(* IEC 61131-3 sources: stverif/testfiles, 5 files *)

(* ---- test.typ ---- *)
TYPE
	My_Struct : STRUCT
		out : INT;
	END_STRUCT;
    Valve : STRUCT
        Value : REAL;
    END_STRUCT;
END_TYPE

(* ---- test.fun ---- *)
FUNCTION I_TO_R : REAL
    VAR_INPUT
        IN : INT;
    END_VAR
END_FUNCTION

(* ---- test.st ---- *)
PROGRAM name_this_program_pls

	// Initialize ControlValues

	FOR n := 1 TO 16 DO
	    k := (45.0 * (k + I_TO_R(n))) / 1000.0;
	END_FOR

	CtrlLEFT  := k;
	CtrlRIGHT := k;

	// Case from the ControlValue with Controller logic action call
  CASE k OF
      1,3,7   :   CtrlLEFT  := a;
      4,6     :   CtrlRIGHT := b;
      ELSE        PosForceCtrl;
  END_CASE

	// Map controller output to hardware
	IF enableCtrlValves.out THEN
	    RightValve.Value    := CtrlLEFT;
	    LeftValve.Value        := CtrlRIGHT;
	ELSE
      ValveCtrl := 0;
  END_IF
END_PROGRAM

(* ---- test.var ---- *)
VAR
    n : INT;
    k : REAL;
    a : REAL;
    b : REAL;
    CtrlLEFT : REAL;
    CtrlRIGHT : REAL;
    enableCtrlValves : My_Struct;
    RightValve : Valve;
    LeftValve : Valve;
    ValveCtrl : INT;
END_VAR

(* ---- test2.st ---- *)
// PosForceCtrl action
ACTION PosForceCtrl :
  IF enableCtrlValves.out THEN
    CtrlLEFT    := CtrlLEFT  + 3.0;
  ELSE
    CtrlRIGHT   := CtrlRIGHT + 3.0;
  END_IF
END_ACTION
